(* IEC 61131-3 sources: PLC-Arduino/PLC/Irrigation-tutorial/pous/functions, 3 files *)

(* ---- eq_State.st ---- *)
FUNCTION eq_State : BOOL
VAR_INPUT
	State1 : irrigation_State;
	State2 : irrigation_State;
END_VAR

if State1 = State2 then
    eq_State := true;
else
    eq_State := false;
end_if;

END_FUNCTION

(* ---- set_State.st ---- *)
FUNCTION set_State : irrigation_State
VAR_INPUT
	State : irrigation_State;
END_VAR

set_State := State;

END_FUNCTION

(* ---- state_To_Num.st ---- *)
FUNCTION state_To_Num : INT
VAR_INPUT
	State : irrigation_State;
END_VAR

if State = Stopped then
    state_To_Num := 0;
elsif State = Running then
    state_To_Num := 1;
elsif State = Manual then
    state_To_Num := 2;
else
    state_To_Num := 3;
end_if;

END_FUNCTION
